{attribute 'Tc2GvlVarNames'}
VAR_GLOBAL
END_VAR

(* stored: Version 1.1.0.1, ProductVersion 3.1.4024.15
   GVL GVAR_Status_and_Alarms: Id {fbb07486-5dc2-4dbe-9458-300792c8594a} *)
